# EPICS autosave request: softGlueApp/Db/scaleOffsetLimit_settings.req
$(P)$(H)SOL-$(N)_S
$(P)$(H)SOL-$(N)_O
$(P)$(H)SOL-$(N)_H
$(P)$(H)SOL-$(N)_L
